// TIA Portal V15.1 export
// export: Created 2022-09-27T21:44:08.9359358Z, ExportSetting WithDefaults, WithReadOnly, DisplayName Totally Integrated Automation Portal, DisplayVersion V15.1 Update 5, DisplayName TIA Portal Openness, DisplayVersion V15.1 Update 5, DisplayName STEP 7 Professional, DisplayVersion V15.1 Update 5, DisplayName WinCC Advanced, DisplayVersion V15.1 Update 5
FUNCTION "Block_1" : Void   // FC1, LAD
{ S7_Optimized_Access := 'TRUE' }
VERSION : 0.1
// stored: AutoNumber true, CodeModifiedDate 2022-09-27T21:42:44.9521673Z, CompileDate 2022-09-27T21:43:15.0961819Z, CreationDate 2022-09-27T21:31:43.3127727Z, HandleErrorsWithinBlock false, InterfaceModifiedDate 2022-09-27T21:32:29.2295254Z, IsConsistent true, IsIECCheckEnabled false, IsKnowHowProtected false, IsWriteProtected false, LibraryConformanceStatus The object is library-conformant., ModifiedDate 2022-09-27T21:42:44.9521673Z, ParameterModified 2022-09-27T21:32:29.2295254Z, PLCSimAdvancedSupport true, SetENOAutomatically False, StructureModified 2022-09-27T21:32:29.2295254Z, UDAEnableTagReadback false
   VAR_INPUT
      Tag1 : Bool;
      Tag2 : Bool;
      Tag3 : Bool;
      Tag4 : Bool;
   END_VAR
   VAR_OUTPUT
      Tag5 : Bool;
      Tag6 : Bool;
   END_VAR
BEGIN

REGION Network 1
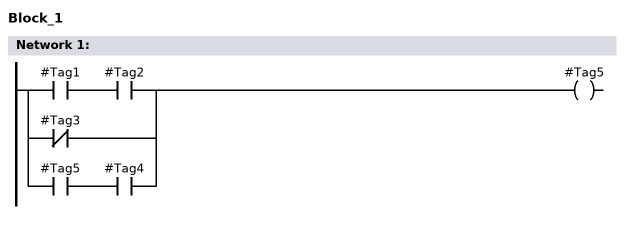
   RUNG wire#powerrail
      Contact( #Tag1 )
      Contact( #Tag2 )
      wire#w1
      Coil( #Tag5 )
   END_RUNG
   RUNG wire#powerrail
      I_Contact( #Tag3 )
   END_RUNG wire#w1
   RUNG wire#powerrail
      Contact( #Tag5 )
      Contact( #Tag4 )
   END_RUNG wire#w1
   // the same network as SCL:
   #Tag5 := (#Tag1 AND #Tag2) OR NOT #Tag3 OR (#Tag5 AND #Tag4);
END_REGION
END_FUNCTION
